INTERFACE I_SessionManager

METHOD PUBLIC CreateSession : T_MAXSTRING
END_METHOD

METHOD PUBLIC DisposeAllSessions
VAR_INPUT
END_VAR
END_METHOD

METHOD PUBLIC IsValidSession : BOOL
VAR_INPUT
	Id : T_MAXSTRING;
END_VAR
END_METHOD

METHOD PUBLIC RefreshSession
VAR_INPUT
	Id : T_MAXSTRING;
END_VAR
END_METHOD

END_INTERFACE

(* stored: Version 1.1.0.1, ProductVersion 3.1.4024.12
   Itf I_SessionManager: Id {80b0fccf-f96c-0ce5-285b-176b28f3ee10}
   Method CreateSession: Id {2ad7424a-a498-09d4-1c07-189bf86ac824}
   Method DisposeAllSessions: Id {c347f40d-dd93-0d19-355a-e4504e28bcd5}
   Method IsValidSession: Id {09668128-ec15-0a35-04c6-efc65b2ad10b}
   Method RefreshSession: Id {e9cc5b66-549e-00e0-2d1c-749b7bff19fd} *)
